(* IEC 61131-3 sources: JaccoSigma/tempclass/Class/CounterRoundTheClock, 1 file *)

(* ---- CounterRoundTheClock.st ---- *)
(*!
<Class
	Name               = "CounterRoundTheClock"
	Revision           = "0.0"
	RealtimeTask       = "false"
	CyclicTask         = "false"
	BackgroundTask     = "false"
	Sigmatek           = "false"
	OSInterface        = "false"
	HighPriority       = "false"
	Automatic          = "false"
	UpdateMode         = "Prescan"
	SharedCommandTable = "true"
	Objectsize         = "(284,120)">
	<Channels>
		<Server Name="AddValue" Visualized="false" Initialize="true" DefValue="1" WriteProtected="false" Retentive="SRam"/>
		<Server Name="OnlyPos" Visualized="false" Initialize="true" DefValue="1" WriteProtected="false" Retentive="SRam"/>
		<Server Name="Range" Visualized="false" Initialize="true" DefValue="1000" WriteProtected="false" Retentive="SRam"/>
		<Server Name="Value" Visualized="false" Initialize="false" WriteProtected="false" Retentive="false"/>
	</Channels>
</Class>
*)
CounterRoundTheClock : CLASS
  //Servers:
	Value 	: SvrChCmd_DINT;
	Range 	: SvrCh_DINT;
	AddValue 	: SvrCh_DINT;
	OnlyPos 	: SvrCh_DINT;
  //Clients:
  //Variables:
  //Functions:

	FUNCTION VIRTUAL GLOBAL Value::Read
		VAR_OUTPUT
			output (EAX) 	: DINT;
		END_VAR;
  //Tables:
	FUNCTION @STD
		VAR_OUTPUT
			ret_code	: CONFSTATES;
		END_VAR;
	FUNCTION GLOBAL TAB @CT_;
END_CLASS;

FUNCTION VIRTUAL GLOBAL CounterRoundTheClock::Value::Read
	VAR_OUTPUT
		output (EAX) 	: DINT;
	END_VAR

  If Range= 0 Then
    // No range so do all
    Value += AddValue;
  Else
    // Within a range
    If AddValue>= 0 Then
      // Count positive
      If Value< Abs( Range) Then
        // Range not reatched
        Value += AddValue;
      else
        // When reatched
        If OnlyPos= 1 Then
          // only positive is 0..range
          Value := 0;
        else
          // -range..0..range
          Value := 0-Abs( Range);
        end_if;
      end_If;
    Else
      // Count negative
      If OnlyPos= 1 Then
        // only positive is range..0
        If Value< 0 Then
          // 0 is not reatched
          Value += AddValue;
        else
          // 0 is reatched. range.. 0
          Value := Abs( Range);
        end_If;
      Else
        // range..0..-range
        If Value> 0-Abs( Range) Then
          // -range not reatched
          Value += AddValue;
        else
          // -range is reatched range..0..-range
          Value := Abs( Range);
        end_If;
      End_If;
    End_If;
  End_If;
  output := Value;

END_FUNCTION
